FUNCTION_BLOCK FirstOrder
VAR_INPUT
	Gain: REAL;
	Tconstant : REAL;
	fBIn   : REAL;
END_VAR
VAR_OUTPUT
	fBOut  : REAL;
END_VAR
VAR
	ssy, Sy   :REAL;
	Tsample: REAL := 0.01;
END_VAR

// Euler Emulation 1st Order with 0.01 sec sampletime.
sy := ( fBIn * Gain / Tconstant ) - ( fBOut / Tconstant ) ;
fBOut := fBout + ( sy * Tsample ) ;

END_FUNCTION_BLOCK

(* stored: Version 1.1.0.1, ProductVersion 3.1.4024.0
   POU FirstOrder: Id {6e10a567-ce2b-41cb-a38e-86d277fe4bcc}, SpecialFunc None *)
